(* CODESYS project FactoryPattern.project

Project tree, tasks and I/O mapping:
  Device : CODESYS Control Win V3, 3S - Smart Software Solutions GmbH, order no. 305021, version 3.5.10.20
    application Application
      libraries: Sheet Metal Factory, 0.0.0.1 (OSB AG)
      task MainTask (cyclic, interval t#20ms, priority 1) calls MY_PRG
  Helper/
    FUNC/
      function incrementInt [ST]
      function decrementInt [ST]
  GVL/
    global variables GVL_CONSTANTS
  program MY_PRG [ST]
  Recipe/
    data type RecipeItem
*)

// Recipe/RecipeItem
TYPE RecipeItem :
STRUCT
	workerType: SMF.WorkerDataType;
	workerData: ARRAY[0..3] OF REAL;
END_STRUCT
END_TYPE

// GVL/GVL_CONSTANTS
VAR_GLOBAL CONSTANT
	MAX_RECIPE_ITEMS: INT := 5;
END_VAR

// MY_PRG
PROGRAM MY_PRG
VAR
	cutterData1: SMF.CutterData := (coords:=[1,1,4,4]);
	cutterData2: SMF.CutterData := (coords:=[1,4,2,4]);
	polisherData1: SMF.PolisherData := (polishDuration:=2000);
	polisherData2: SMF.PolisherData := (polishDuration:=3500);
	idleData: SMF.IdleData;
	
	recipe: ARRAY[1..5] OF SMF.IWorkerData := [ cutterData1, polisherData1, cutterData2, polisherData2, idleData];
	
	sequenceFactory: SMF.SequenceFactory;
		
	actWorker: SMF.IWorker;
	actWorkerType : SMF.WorkerDataType;
	
	xDestroy: BOOL;
	isInit: BOOL;
END_VAR

IF NOT isInit THEN
	actWorker := sequenceFactory.generateSequence(recipe);
	
	isInit := TRUE; 
END_IF

IF actWorker <> 0  THEN
	actWorker := actWorker.process();			//let the workers do their work
	actWorkerType := actWorker.workerType;		//read worker type just to see them change
END_IF


//cleanup instances	
IF xDestroy THEN
	sequenceFactory.cleanUp();
	actWorker := 0;
	
	xDestroy := FALSE;
END_IF

END_PROGRAM

// Helper/FUNC/incrementInt
FUNCTION incrementInt : bool
VAR_INPUT
	var2Increment : REFERENCE TO INT;
	
END_VAR
VAR
END_VAR

IF var2Increment < 16#7FFF THEN
	var2Increment := var2Increment + 1;
END_IF

END_FUNCTION

// Helper/FUNC/decrementInt
FUNCTION decrementInt : bool
VAR_INPUT
	var2Decrement : REFERENCE TO INT;
END_VAR
VAR
END_VAR

IF var2Decrement > -32768 THEN
	var2Decrement := var2Decrement - 1;
END_IF

END_FUNCTION
